{attribute addProperty BoxType "EK1122-0000-0018"}
{attribute addProperty Id "Beckhoff_ER2xxxsub_EK1100EK1100_179A0949162A_0001_ER2008_0001_0018ER2008_A854BE6D8110.125A_0002_ER2008_0001_0019ER2008_A854BE6D8110.125A_0003_ER2008_0002_0018ER2008_A854BE6D8110.125A_0004_ER2008_0002_0019ER2008_A854BE6D8110.125A_0005_ER2008_0022_0017ER2008_A854BE6D8110.125A_0006_ER2008_0022_0018ER2008_A854BE6D8110.125A_0007_ER2028_0001_0017ER2028_A854BE6D8110.125A_0008_ER2028_0001_0018ER2028_A854BE6D8110.125A_0009_ER2028_0002_0018ER2028_A854BE6D8110.125A_0010_ER2028_0002_0019ER2028_A854BE6D8110.125A_0011_ER2028_1032_0016ER2028_A854BE6D8110.125A_0012_ER2038_0001_0017ER2038_9444C9D314618.25A_0013_ER2038_0001_0018ER2038_9444C9D314618.25A_0014_ER2038_0002_0017ER2038_9444C9D314618.25A_0015_ER2038_0002_0018ER2038_9444C9D314618.25A_0016_ER2308_0001_0018ER2308_97B4DD118210.25A_0017_ER2308_0001_0019ER2308_97B4DD118210.25A_0018_ER2308_0002_0018ER2308_97B4DD118210.25A_0019_ER2308_0002_0019ER2308_97B4DD118210.25A_0020_ER2318_0001_0018ER2318_97B4DD118210.25A_0021_ER2318_0001_0019ER2318_97B4DD118210.25A_0022_ER2318_0002_0018ER2318_97B4DD118210.25A_0023_ER2318_0002_0019ER2318_97B4DD118210.25A_0024_ER2328_0001_0017ER2328_97B4DD118210.25A_0025_ER2328_0001_0018ER2328_97B4DD118210.25A_0026_ER2328_0002_0018ER2328_97B4DD118210.25A_0027_ER2328_0002_0019ER2328_97B4DD118210.25A_0028_ER2338_0001_0022ER2338_538B459D14618.25A_0029_ER2338_0001_0023ER2338_538B459D14618.25A_0030_ER2338_0002_0022ER2338_538B459D14618.25A_0031_ER2338_0002_0023ER2338_538B459D14618.25A_0032_ER2338_1001_0017ER2338_538B459D14618.25A_0033_ER2338_1001_0018ER2338_538B459D14618.25A_0034_ER2338_1002_0017ER2338_538B459D14618.25A_0035_ER2338_1002_0018ER2338_538B459D14618.25A_0036_ER2339_0021_0018ER2339_BBE0865932240.25A_0037_ER2339_0021_0019ER2339_9219B49827434.25A_0038_ER2339_0022_0018ER2339_9219B49827434.25A_0039_ER2339_0022_0019ER2339_9219B49827434.25A_0040_ER2349_0021_0017ER2349_9219B49827434.25A_0041_ER2349_0021_0018ER2349_9219B49827434.25A_0042_ER2349_0022_0017ER2349_9219B49827434.25A_0043_ER2349_0022_0018ER2349_9219B49827434.25A_0044_ER2624_0002_0018ER2624_4E3C7537496.125A_0045_ER2624_0002_0019ER2624_4E3C7537496.125A_0046_ER2809_0021_0017ER2809_859F43D214518.125A_0047_ER2809_0021_0018ER2809_859F43D214518.125A_0048_ER2809_0022_0016ER2809_859F43D214518.125A_0049_ER2809_0022_0017ER2809_859F43D214518.125A_0050_ER2809_0022_0018ER2809_859F43D214518.125"}
{attribute addProperty CRC "3261673935"}
{attribute addProperty SizeInBites "6706"}
{attribute addProperty SizeInBytes "838.25"}
TYPE Beckhoff_ER2xxxEK1122_C26931CF EXTENDS EK1122_179A0949 :
STRUCT
	{attribute addProperty Name "Beckhoff_ER2xxxsub_EK1100"}
	Beckhoff_ER2xxxsub_EK1100 : EK1100_179A0949;
	{attribute addProperty Name "A_0001_ER2008_0001_0018"}
	A_0001_ER2008_0001_0018 : ER2008_A854BE6D;
	{attribute addProperty Name "A_0002_ER2008_0001_0019"}
	A_0002_ER2008_0001_0019 : ER2008_A854BE6D;
	{attribute addProperty Name "A_0003_ER2008_0002_0018"}
	A_0003_ER2008_0002_0018 : ER2008_A854BE6D;
	{attribute addProperty Name "A_0004_ER2008_0002_0019"}
	A_0004_ER2008_0002_0019 : ER2008_A854BE6D;
	{attribute addProperty Name "A_0005_ER2008_0022_0017"}
	A_0005_ER2008_0022_0017 : ER2008_A854BE6D;
	{attribute addProperty Name "A_0006_ER2008_0022_0018"}
	A_0006_ER2008_0022_0018 : ER2008_A854BE6D;
	{attribute addProperty Name "A_0007_ER2028_0001_0017"}
	A_0007_ER2028_0001_0017 : ER2028_A854BE6D;
	{attribute addProperty Name "A_0008_ER2028_0001_0018"}
	A_0008_ER2028_0001_0018 : ER2028_A854BE6D;
	{attribute addProperty Name "A_0009_ER2028_0002_0018"}
	A_0009_ER2028_0002_0018 : ER2028_A854BE6D;
	{attribute addProperty Name "A_0010_ER2028_0002_0019"}
	A_0010_ER2028_0002_0019 : ER2028_A854BE6D;
	{attribute addProperty Name "A_0011_ER2028_1032_0016"}
	A_0011_ER2028_1032_0016 : ER2028_A854BE6D;
	{attribute addProperty Name "A_0012_ER2038_0001_0017"}
	A_0012_ER2038_0001_0017 : ER2038_9444C9D3;
	{attribute addProperty Name "A_0013_ER2038_0001_0018"}
	A_0013_ER2038_0001_0018 : ER2038_9444C9D3;
	{attribute addProperty Name "A_0014_ER2038_0002_0017"}
	A_0014_ER2038_0002_0017 : ER2038_9444C9D3;
	{attribute addProperty Name "A_0015_ER2038_0002_0018"}
	A_0015_ER2038_0002_0018 : ER2038_9444C9D3;
	{attribute addProperty Name "A_0016_ER2308_0001_0018"}
	A_0016_ER2308_0001_0018 : ER2308_97B4DD11;
	{attribute addProperty Name "A_0017_ER2308_0001_0019"}
	A_0017_ER2308_0001_0019 : ER2308_97B4DD11;
	{attribute addProperty Name "A_0018_ER2308_0002_0018"}
	A_0018_ER2308_0002_0018 : ER2308_97B4DD11;
	{attribute addProperty Name "A_0019_ER2308_0002_0019"}
	A_0019_ER2308_0002_0019 : ER2308_97B4DD11;
	{attribute addProperty Name "A_0020_ER2318_0001_0018"}
	A_0020_ER2318_0001_0018 : ER2318_97B4DD11;
	{attribute addProperty Name "A_0021_ER2318_0001_0019"}
	A_0021_ER2318_0001_0019 : ER2318_97B4DD11;
	{attribute addProperty Name "A_0022_ER2318_0002_0018"}
	A_0022_ER2318_0002_0018 : ER2318_97B4DD11;
	{attribute addProperty Name "A_0023_ER2318_0002_0019"}
	A_0023_ER2318_0002_0019 : ER2318_97B4DD11;
	{attribute addProperty Name "A_0024_ER2328_0001_0017"}
	A_0024_ER2328_0001_0017 : ER2328_97B4DD11;
	{attribute addProperty Name "A_0025_ER2328_0001_0018"}
	A_0025_ER2328_0001_0018 : ER2328_97B4DD11;
	{attribute addProperty Name "A_0026_ER2328_0002_0018"}
	A_0026_ER2328_0002_0018 : ER2328_97B4DD11;
	{attribute addProperty Name "A_0027_ER2328_0002_0019"}
	A_0027_ER2328_0002_0019 : ER2328_97B4DD11;
	{attribute addProperty Name "A_0028_ER2338_0001_0022"}
	A_0028_ER2338_0001_0022 : ER2338_538B459D;
	{attribute addProperty Name "A_0029_ER2338_0001_0023"}
	A_0029_ER2338_0001_0023 : ER2338_538B459D;
	{attribute addProperty Name "A_0030_ER2338_0002_0022"}
	A_0030_ER2338_0002_0022 : ER2338_538B459D;
	{attribute addProperty Name "A_0031_ER2338_0002_0023"}
	A_0031_ER2338_0002_0023 : ER2338_538B459D;
	{attribute addProperty Name "A_0032_ER2338_1001_0017"}
	A_0032_ER2338_1001_0017 : ER2338_538B459D;
	{attribute addProperty Name "A_0033_ER2338_1001_0018"}
	A_0033_ER2338_1001_0018 : ER2338_538B459D;
	{attribute addProperty Name "A_0034_ER2338_1002_0017"}
	A_0034_ER2338_1002_0017 : ER2338_538B459D;
	{attribute addProperty Name "A_0035_ER2338_1002_0018"}
	A_0035_ER2338_1002_0018 : ER2338_538B459D;
	{attribute addProperty Name "A_0036_ER2339_0021_0018"}
	A_0036_ER2339_0021_0018 : ER2339_BBE08659;
	{attribute addProperty Name "A_0037_ER2339_0021_0019"}
	A_0037_ER2339_0021_0019 : ER2339_9219B498;
	{attribute addProperty Name "A_0038_ER2339_0022_0018"}
	A_0038_ER2339_0022_0018 : ER2339_9219B498;
	{attribute addProperty Name "A_0039_ER2339_0022_0019"}
	A_0039_ER2339_0022_0019 : ER2339_9219B498;
	{attribute addProperty Name "A_0040_ER2349_0021_0017"}
	A_0040_ER2349_0021_0017 : ER2349_9219B498;
	{attribute addProperty Name "A_0041_ER2349_0021_0018"}
	A_0041_ER2349_0021_0018 : ER2349_9219B498;
	{attribute addProperty Name "A_0042_ER2349_0022_0017"}
	A_0042_ER2349_0022_0017 : ER2349_9219B498;
	{attribute addProperty Name "A_0043_ER2349_0022_0018"}
	A_0043_ER2349_0022_0018 : ER2349_9219B498;
	{attribute addProperty Name "A_0044_ER2624_0002_0018"}
	A_0044_ER2624_0002_0018 : ER2624_4E3C7537;
	{attribute addProperty Name "A_0045_ER2624_0002_0019"}
	A_0045_ER2624_0002_0019 : ER2624_4E3C7537;
	{attribute addProperty Name "A_0046_ER2809_0021_0017"}
	A_0046_ER2809_0021_0017 : ER2809_859F43D2;
	{attribute addProperty Name "A_0047_ER2809_0021_0018"}
	A_0047_ER2809_0021_0018 : ER2809_859F43D2;
	{attribute addProperty Name "A_0048_ER2809_0022_0016"}
	A_0048_ER2809_0022_0016 : ER2809_859F43D2;
	{attribute addProperty Name "A_0049_ER2809_0022_0017"}
	A_0049_ER2809_0022_0017 : ER2809_859F43D2;
	{attribute addProperty Name "A_0050_ER2809_0022_0018"}
	A_0050_ER2809_0022_0018 : ER2809_859F43D2;
END_STRUCT
END_TYPE

(* stored: Version 1.2.0.0, ProductVersion 3.1.4024.9
   DUT Beckhoff_ER2xxxEK1122_C26931CF: Id {61e6dc27-f606-42e1-950e-5e5bb1246e3c} *)
